//     Enc/Inputs/In/nState2 @bit 5 <-> ENC Status compact Channel 1/Status/Sync error
//     Enc/Inputs/In/nState2 @bit 5 <-> ENC Status compact Channel 2/Status/Sync error
//     Enc/Inputs/In/nState2 @bit 7 <-> ENC Status compact Channel 1/Status/TxPDO Toggle
//     Enc/Inputs/In/nState2 @bit 7 <-> ENC Status compact Channel 2/Status/TxPDO Toggle
//     Enc/Inputs/In/nState4 @bit 1 <-> WcState/InputToggle
//     Enc/Inputs/In/nState4 <-> WcState/WcState
//     Enc/Outputs/Out/nCtrl1 @bit 3 <-> ENC Control compact Channel 1/Control/Enable latch extern on negative edge
//     Enc/Outputs/Out/nCtrl1 @bit 3 <-> ENC Control compact Channel 2/Control/Enable latch extern on negative edge
//     Enc/Outputs/Out/nCtrl1 @bit 1 <-> ENC Control compact Channel 1/Control/Enable latch extern on positive edge
//     Enc/Outputs/Out/nCtrl1 @bit 1 <-> ENC Control compact Channel 2/Control/Enable latch extern on positive edge
//     Enc/Outputs/Out/nCtrl1 @bit 2 <-> ENC Control compact Channel 1/Control/Set counter
//     Enc/Outputs/Out/nCtrl1 @bit 2 <-> ENC Control compact Channel 2/Control/Set counter
//     Enc/Outputs/Out/nDataOut1[0] <-> ENC Control compact Channel 1/Set counter value
//     Enc/Outputs/Out/nDataOut1[0] <-> ENC Control compact Channel 2/Set counter value
//   NC-Task 1 SAF/Axes/Axis 1 <-> Long-CarryDrop (EtherCAT)/Long-Straight 1 (EP7342-0002)
//     Drive/Inputs/In/nState1 @bit 3 <-> DCM Status Channel 1/Status/Error
//     Drive/Inputs/In/nState1 @bit 5 <-> DCM Status Channel 1/Status/Moving negative
//     Drive/Inputs/In/nState1 @bit 4 <-> DCM Status Channel 1/Status/Moving positive
//     Drive/Inputs/In/nState1 @bit 1 <-> DCM Status Channel 1/Status/Ready
//     Drive/Inputs/In/nState1 <-> DCM Status Channel 1/Status/Ready to enable
//     Drive/Inputs/In/nState1 @bit 6 <-> DCM Status Channel 1/Status/Torque reduced
//     Drive/Inputs/In/nState1 @bit 2 <-> DCM Status Channel 1/Status/Warning
//     Drive/Inputs/In/nState2 @bit 3 <-> DCM Status Channel 1/Status/Digital input 1
//     Drive/Inputs/In/nState2 @bit 4 <-> DCM Status Channel 1/Status/Digital input 2
//     Drive/Inputs/In/nState2 @bit 5 <-> DCM Status Channel 1/Status/Sync error
//     Drive/Inputs/In/nState2 @bit 7 <-> DCM Status Channel 1/Status/TxPDO Toggle
//     Drive/Inputs/In/nState4 @bit 1 <-> WcState/InputToggle
//     Drive/Inputs/In/nState4 <-> WcState/WcState
//     Drive/Outputs/Out/nCtrl1 <-> DCM Control Channel 1/Control/Enable
//     Drive/Outputs/Out/nCtrl1 @bit 2 <-> DCM Control Channel 1/Control/Reduce torque
//     Drive/Outputs/Out/nCtrl1 @bit 1 <-> DCM Control Channel 1/Control/Reset
//     Drive/Outputs/Out/nDataOut2[0] <-> DCM Velocity Channel 1/Velocity
//     Enc/Inputs/In/nDataIn1[0] <-> ENC Status compact Channel 1/Counter value
//     Enc/Inputs/In/nDataIn2[0] <-> ENC Status compact Channel 1/Latch value
//     Enc/Inputs/In/nState1 @bit 4 <-> ENC Status compact Channel 1/Status/Counter overflow
//     Enc/Inputs/In/nState1 @bit 3 <-> ENC Status compact Channel 1/Status/Counter underflow
//     Enc/Inputs/In/nState1 @bit 7 <-> ENC Status compact Channel 1/Status/Extrapolation stall
//     Enc/Inputs/In/nState1 @bit 1 <-> ENC Status compact Channel 1/Status/Latch extern valid
//     Enc/Inputs/In/nState1 @bit 2 <-> ENC Status compact Channel 1/Status/Set counter done
//     Enc/Inputs/In/nState2 @bit 4 <-> ENC Status compact Channel 1/Status/Status of extern latch
//     Enc/Inputs/In/nState2 <-> ENC Status compact Channel 1/Status/Status of input A
//     Enc/Inputs/In/nState2 @bit 1 <-> ENC Status compact Channel 1/Status/Status of input B
//     Enc/Inputs/In/nState2 @bit 5 <-> ENC Status compact Channel 1/Status/Sync error
//     Enc/Inputs/In/nState2 @bit 7 <-> ENC Status compact Channel 1/Status/TxPDO Toggle
//     Enc/Inputs/In/nState4 @bit 1 <-> WcState/InputToggle
//     Enc/Inputs/In/nState4 <-> WcState/WcState
//     Enc/Outputs/Out/nCtrl1 @bit 3 <-> ENC Control compact Channel 1/Control/Enable latch extern on negative edge
//     Enc/Outputs/Out/nCtrl1 @bit 1 <-> ENC Control compact Channel 1/Control/Enable latch extern on positive edge
//     Enc/Outputs/Out/nCtrl1 @bit 2 <-> ENC Control compact Channel 1/Control/Set counter
//     Enc/Outputs/Out/nDataOut1[0] <-> ENC Control compact Channel 1/Set counter value
//   NC-Task 1 SAF/Axes/Axis 1 <-> Untitled1/Untitled1 Instance
//     Inputs/FromPlc <-> PlcTask Outputs/MAIN.stAxis1.PlcToNc
//     Outputs/ToPlc <-> PlcTask Inputs/MAIN.stAxis1.NcToPlc
//   NC-Task 1 SAF/Axes/Axis 2 <-> Long-CarryDrop (EtherCAT)/Long-Straight 1 (EP7342-0002)
//     Drive/Inputs/In/nState1 @bit 3 <-> DCM Status Channel 2/Status/Error
//     Drive/Inputs/In/nState1 @bit 5 <-> DCM Status Channel 2/Status/Moving negative
//     Drive/Inputs/In/nState1 @bit 4 <-> DCM Status Channel 2/Status/Moving positive
//     Drive/Inputs/In/nState1 @bit 1 <-> DCM Status Channel 2/Status/Ready
//     Drive/Inputs/In/nState1 <-> DCM Status Channel 2/Status/Ready to enable
//     Drive/Inputs/In/nState1 @bit 6 <-> DCM Status Channel 2/Status/Torque reduced
//     Drive/Inputs/In/nState1 @bit 2 <-> DCM Status Channel 2/Status/Warning
//     Drive/Inputs/In/nState2 @bit 3 <-> DCM Status Channel 2/Status/Digital input 1
//     Drive/Inputs/In/nState2 @bit 4 <-> DCM Status Channel 2/Status/Digital input 2
//     Drive/Inputs/In/nState2 @bit 5 <-> DCM Status Channel 2/Status/Sync error
//     Drive/Inputs/In/nState2 @bit 7 <-> DCM Status Channel 2/Status/TxPDO Toggle
//     Drive/Inputs/In/nState4 @bit 1 <-> WcState/InputToggle
//     Drive/Inputs/In/nState4 <-> WcState/WcState
//     Drive/Outputs/Out/nCtrl1 <-> DCM Control Channel 2/Control/Enable
//     Drive/Outputs/Out/nCtrl1 @bit 2 <-> DCM Control Channel 2/Control/Reduce torque
//     Drive/Outputs/Out/nCtrl1 @bit 1 <-> DCM Control Channel 2/Control/Reset
//     Drive/Outputs/Out/nDataOut2[0] <-> DCM Velocity Channel 2/Velocity
//     Enc/Inputs/In/nDataIn1[0] <-> ENC Status compact Channel 2/Counter value
//     Enc/Inputs/In/nDataIn2[0] <-> ENC Status compact Channel 2/Latch value
//     Enc/Inputs/In/nState1 @bit 4 <-> ENC Status compact Channel 2/Status/Counter overflow
//     Enc/Inputs/In/nState1 @bit 3 <-> ENC Status compact Channel 2/Status/Counter underflow
//     Enc/Inputs/In/nState1 @bit 7 <-> ENC Status compact Channel 2/Status/Extrapolation stall
//     Enc/Inputs/In/nState1 @bit 1 <-> ENC Status compact Channel 2/Status/Latch extern valid
//     Enc/Inputs/In/nState1 @bit 2 <-> ENC Status compact Channel 2/Status/Set counter done
//     Enc/Inputs/In/nState2 @bit 4 <-> ENC Status compact Channel 2/Status/Status of extern latch
//     Enc/Inputs/In/nState2 <-> ENC Status compact Channel 2/Status/Status of input A
//     Enc/Inputs/In/nState2 @bit 1 <-> ENC Status compact Channel 2/Status/Status of input B
//     Enc/Inputs/In/nState2 @bit 5 <-> ENC Status compact Channel 2/Status/Sync error
//     Enc/Inputs/In/nState2 @bit 7 <-> ENC Status compact Channel 2/Status/TxPDO Toggle
//     Enc/Inputs/In/nState4 @bit 1 <-> WcState/InputToggle
//     Enc/Inputs/In/nState4 <-> WcState/WcState
//     Enc/Outputs/Out/nCtrl1 @bit 3 <-> ENC Control compact Channel 2/Control/Enable latch extern on negative edge
//     Enc/Outputs/Out/nCtrl1 @bit 1 <-> ENC Control compact Channel 2/Control/Enable latch extern on positive edge
//     Enc/Outputs/Out/nCtrl1 @bit 2 <-> ENC Control compact Channel 2/Control/Set counter
//     Enc/Outputs/Out/nDataOut1[0] <-> ENC Control compact Channel 2/Set counter value
//   NC-Task 1 SAF/Axes/Axis 2 <-> Untitled1/Untitled1 Instance
//     Inputs/FromPlc <-> PlcTask Outputs/MAIN.stAxis2.PlcToNc
//     Outputs/ToPlc <-> PlcTask Inputs/MAIN.stAxis2.NcToPlc
//   NC-Task 1 SAF/Axes/Axis 3 <-> Long-CarryDrop (EtherCAT)/Long-Straight 2 (EP7342-0002)
//     Drive/Inputs/In/nState1 @bit 3 <-> DCM Status Channel 1/Status/Error
//     Drive/Inputs/In/nState1 @bit 5 <-> DCM Status Channel 1/Status/Moving negative
//     Drive/Inputs/In/nState1 @bit 4 <-> DCM Status Channel 1/Status/Moving positive
//     Drive/Inputs/In/nState1 @bit 1 <-> DCM Status Channel 1/Status/Ready
//     Drive/Inputs/In/nState1 <-> DCM Status Channel 1/Status/Ready to enable
//     Drive/Inputs/In/nState1 @bit 6 <-> DCM Status Channel 1/Status/Torque reduced
//     Drive/Inputs/In/nState1 @bit 2 <-> DCM Status Channel 1/Status/Warning
//     Drive/Inputs/In/nState2 @bit 3 <-> DCM Status Channel 1/Status/Digital input 1
//     Drive/Inputs/In/nState2 @bit 4 <-> DCM Status Channel 1/Status/Digital input 2
//     Drive/Inputs/In/nState2 @bit 5 <-> DCM Status Channel 1/Status/Sync error
//     Drive/Inputs/In/nState2 @bit 7 <-> DCM Status Channel 1/Status/TxPDO Toggle
//     Drive/Inputs/In/nState4 @bit 1 <-> WcState/InputToggle
//     Drive/Inputs/In/nState4 <-> WcState/WcState
//     Drive/Outputs/Out/nCtrl1 <-> DCM Control Channel 1/Control/Enable
//     Drive/Outputs/Out/nCtrl1 @bit 2 <-> DCM Control Channel 1/Control/Reduce torque
//     Drive/Outputs/Out/nCtrl1 @bit 1 <-> DCM Control Channel 1/Control/Reset
//     Drive/Outputs/Out/nDataOut2[0] <-> DCM Velocity Channel 1/Velocity
//     Enc/Inputs/In/nDataIn1[0] <-> ENC Status compact Channel 1/Counter value
//     Enc/Inputs/In/nDataIn2[0] <-> ENC Status compact Channel 1/Latch value
//     Enc/Inputs/In/nState1 @bit 4 <-> ENC Status compact Channel 1/Status/Counter overflow
//     Enc/Inputs/In/nState1 @bit 3 <-> ENC Status compact Channel 1/Status/Counter underflow
//     Enc/Inputs/In/nState1 @bit 7 <-> ENC Status compact Channel 1/Status/Extrapolation stall
//     Enc/Inputs/In/nState1 @bit 1 <-> ENC Status compact Channel 1/Status/Latch extern valid
//     Enc/Inputs/In/nState1 @bit 2 <-> ENC Status compact Channel 1/Status/Set counter done
//     Enc/Inputs/In/nState2 @bit 4 <-> ENC Status compact Channel 1/Status/Status of extern latch
//     Enc/Inputs/In/nState2 <-> ENC Status compact Channel 1/Status/Status of input A
//     Enc/Inputs/In/nState2 @bit 1 <-> ENC Status compact Channel 1/Status/Status of input B
//     Enc/Inputs/In/nState2 @bit 5 <-> ENC Status compact Channel 1/Status/Sync error
//     Enc/Inputs/In/nState2 @bit 7 <-> ENC Status compact Channel 1/Status/TxPDO Toggle
//     Enc/Inputs/In/nState4 @bit 1 <-> WcState/InputToggle
//     Enc/Inputs/In/nState4 <-> WcState/WcState
//     Enc/Outputs/Out/nCtrl1 @bit 3 <-> ENC Control compact Channel 1/Control/Enable latch extern on negative edge
//     Enc/Outputs/Out/nCtrl1 @bit 1 <-> ENC Control compact Channel 1/Control/Enable latch extern on positive edge
//     Enc/Outputs/Out/nCtrl1 @bit 2 <-> ENC Control compact Channel 1/Control/Set counter
//     Enc/Outputs/Out/nDataOut1[0] <-> ENC Control compact Channel 1/Set counter value
//   NC-Task 1 SAF/Axes/Axis 3 <-> Untitled1/Untitled1 Instance
//     Inputs/FromPlc <-> PlcTask Outputs/MAIN.stAxis3.PlcToNc
//     Outputs/ToPlc <-> PlcTask Inputs/MAIN.stAxis3.NcToPlc
//   NC-Task 1 SAF/Axes/Axis 4 <-> Long-CarryDrop (EtherCAT)/Long-Straight 2 (EP7342-0002)
//     Drive/Inputs/In/nState1 @bit 3 <-> DCM Status Channel 2/Status/Error
//     Drive/Inputs/In/nState1 @bit 5 <-> DCM Status Channel 2/Status/Moving negative
//     Drive/Inputs/In/nState1 @bit 4 <-> DCM Status Channel 2/Status/Moving positive
//     Drive/Inputs/In/nState1 @bit 1 <-> DCM Status Channel 2/Status/Ready
//     Drive/Inputs/In/nState1 <-> DCM Status Channel 2/Status/Ready to enable
//     Drive/Inputs/In/nState1 @bit 6 <-> DCM Status Channel 2/Status/Torque reduced
//     Drive/Inputs/In/nState1 @bit 2 <-> DCM Status Channel 2/Status/Warning
//     Drive/Inputs/In/nState2 @bit 3 <-> DCM Status Channel 2/Status/Digital input 1
//     Drive/Inputs/In/nState2 @bit 4 <-> DCM Status Channel 2/Status/Digital input 2
//     Drive/Inputs/In/nState2 @bit 5 <-> DCM Status Channel 2/Status/Sync error
//     Drive/Inputs/In/nState2 @bit 7 <-> DCM Status Channel 2/Status/TxPDO Toggle
//     Drive/Inputs/In/nState4 @bit 1 <-> WcState/InputToggle
//     Drive/Inputs/In/nState4 <-> WcState/WcState
//     Drive/Outputs/Out/nCtrl1 <-> DCM Control Channel 2/Control/Enable
//     Drive/Outputs/Out/nCtrl1 @bit 2 <-> DCM Control Channel 2/Control/Reduce torque
//     Drive/Outputs/Out/nCtrl1 @bit 1 <-> DCM Control Channel 2/Control/Reset
//     Drive/Outputs/Out/nDataOut2[0] <-> DCM Velocity Channel 2/Velocity
//     Enc/Inputs/In/nDataIn1[0] <-> ENC Status compact Channel 2/Counter value
//     Enc/Inputs/In/nDataIn2[0] <-> ENC Status compact Channel 2/Latch value
//     Enc/Inputs/In/nState1 @bit 4 <-> ENC Status compact Channel 2/Status/Counter overflow
//     Enc/Inputs/In/nState1 @bit 3 <-> ENC Status compact Channel 2/Status/Counter underflow
//     Enc/Inputs/In/nState1 @bit 7 <-> ENC Status compact Channel 2/Status/Extrapolation stall
//     Enc/Inputs/In/nState1 @bit 1 <-> ENC Status compact Channel 2/Status/Latch extern valid
//     Enc/Inputs/In/nState1 @bit 2 <-> ENC Status compact Channel 2/Status/Set counter done
//     Enc/Inputs/In/nState2 @bit 4 <-> ENC Status compact Channel 2/Status/Status of extern latch
//     Enc/Inputs/In/nState2 <-> ENC Status compact Channel 2/Status/Status of input A
//     Enc/Inputs/In/nState2 @bit 1 <-> ENC Status compact Channel 2/Status/Status of input B
//     Enc/Inputs/In/nState2 @bit 5 <-> ENC Status compact Channel 2/Status/Sync error
//     Enc/Inputs/In/nState2 @bit 7 <-> ENC Status compact Channel 2/Status/TxPDO Toggle
//     Enc/Inputs/In/nState4 @bit 1 <-> WcState/InputToggle
//     Enc/Inputs/In/nState4 <-> WcState/WcState
//     Enc/Outputs/Out/nCtrl1 @bit 3 <-> ENC Control compact Channel 2/Control/Enable latch extern on negative edge
//     Enc/Outputs/Out/nCtrl1 @bit 1 <-> ENC Control compact Channel 2/Control/Enable latch extern on positive edge
//     Enc/Outputs/Out/nCtrl1 @bit 2 <-> ENC Control compact Channel 2/Control/Set counter
//     Enc/Outputs/Out/nDataOut1[0] <-> ENC Control compact Channel 2/Set counter value
//   NC-Task 1 SAF/Axes/Axis 4 <-> Untitled1/Untitled1 Instance
//     Inputs/FromPlc <-> PlcTask Outputs/MAIN.stAxis4.PlcToNc
//     Outputs/ToPlc <-> PlcTask Inputs/MAIN.stAxis4.NcToPlc
//   NC-Task 1 SAF/Axes/Axis 5 <-> Long-CarryDrop (EtherCAT)/Short-Straight 1 (EP7342-0002)
//     Drive/Inputs/In/nState1 @bit 3 <-> DCM Status Channel 1/Status/Error
//     Drive/Inputs/In/nState1 @bit 5 <-> DCM Status Channel 1/Status/Moving negative
//     Drive/Inputs/In/nState1 @bit 4 <-> DCM Status Channel 1/Status/Moving positive
//     Drive/Inputs/In/nState1 @bit 1 <-> DCM Status Channel 1/Status/Ready
//     Drive/Inputs/In/nState1 <-> DCM Status Channel 1/Status/Ready to enable
//     Drive/Inputs/In/nState1 @bit 6 <-> DCM Status Channel 1/Status/Torque reduced
//     Drive/Inputs/In/nState1 @bit 2 <-> DCM Status Channel 1/Status/Warning
//     Drive/Inputs/In/nState2 @bit 3 <-> DCM Status Channel 1/Status/Digital input 1
//     Drive/Inputs/In/nState2 @bit 4 <-> DCM Status Channel 1/Status/Digital input 2
//     Drive/Inputs/In/nState2 @bit 5 <-> DCM Status Channel 1/Status/Sync error
//     Drive/Inputs/In/nState2 @bit 7 <-> DCM Status Channel 1/Status/TxPDO Toggle
//     Drive/Inputs/In/nState4 @bit 1 <-> WcState/InputToggle
//     Drive/Inputs/In/nState4 <-> WcState/WcState
//     Drive/Outputs/Out/nCtrl1 <-> DCM Control Channel 1/Control/Enable
//     Drive/Outputs/Out/nCtrl1 @bit 2 <-> DCM Control Channel 1/Control/Reduce torque
//     Drive/Outputs/Out/nCtrl1 @bit 1 <-> DCM Control Channel 1/Control/Reset
//     Drive/Outputs/Out/nDataOut2[0] <-> DCM Velocity Channel 1/Velocity
//     Enc/Inputs/In/nDataIn1[0] <-> ENC Status compact Channel 1/Counter value
//     Enc/Inputs/In/nDataIn2[0] <-> ENC Status compact Channel 1/Latch value
//     Enc/Inputs/In/nState1 @bit 4 <-> ENC Status compact Channel 1/Status/Counter overflow
//     Enc/Inputs/In/nState1 @bit 3 <-> ENC Status compact Channel 1/Status/Counter underflow
//     Enc/Inputs/In/nState1 @bit 7 <-> ENC Status compact Channel 1/Status/Extrapolation stall
//     Enc/Inputs/In/nState1 @bit 1 <-> ENC Status compact Channel 1/Status/Latch extern valid
//     Enc/Inputs/In/nState1 @bit 2 <-> ENC Status compact Channel 1/Status/Set counter done
//     Enc/Inputs/In/nState2 @bit 4 <-> ENC Status compact Channel 1/Status/Status of extern latch
//     Enc/Inputs/In/nState2 <-> ENC Status compact Channel 1/Status/Status of input A
//     Enc/Inputs/In/nState2 @bit 1 <-> ENC Status compact Channel 1/Status/Status of input B
//     Enc/Inputs/In/nState2 @bit 5 <-> ENC Status compact Channel 1/Status/Sync error
//     Enc/Inputs/In/nState2 @bit 7 <-> ENC Status compact Channel 1/Status/TxPDO Toggle
//     Enc/Inputs/In/nState4 @bit 1 <-> WcState/InputToggle
//     Enc/Inputs/In/nState4 <-> WcState/WcState
//     Enc/Outputs/Out/nCtrl1 @bit 3 <-> ENC Control compact Channel 1/Control/Enable latch extern on negative edge
//     Enc/Outputs/Out/nCtrl1 @bit 1 <-> ENC Control compact Channel 1/Control/Enable latch extern on positive edge
//     Enc/Outputs/Out/nCtrl1 @bit 2 <-> ENC Control compact Channel 1/Control/Set counter
//     Enc/Outputs/Out/nDataOut1[0] <-> ENC Control compact Channel 1/Set counter value
//   NC-Task 1 SAF/Axes/Axis 5 <-> Untitled1/Untitled1 Instance
//     Inputs/FromPlc <-> PlcTask Outputs/MAIN.stAxis5.PlcToNc
//     Outputs/ToPlc <-> PlcTask Inputs/MAIN.stAxis5.NcToPlc
//   NC-Task 1 SAF/Axes/Axis 6 <-> Long-CarryDrop (EtherCAT)/Short-Straight 1 (EP7342-0002)
//     Drive/Inputs/In/nState1 @bit 3 <-> DCM Status Channel 2/Status/Error
//     Drive/Inputs/In/nState1 @bit 5 <-> DCM Status Channel 2/Status/Moving negative
//     Drive/Inputs/In/nState1 @bit 4 <-> DCM Status Channel 2/Status/Moving positive
//     Drive/Inputs/In/nState1 @bit 1 <-> DCM Status Channel 2/Status/Ready
//     Drive/Inputs/In/nState1 <-> DCM Status Channel 2/Status/Ready to enable
//     Drive/Inputs/In/nState1 @bit 6 <-> DCM Status Channel 2/Status/Torque reduced
//     Drive/Inputs/In/nState1 @bit 2 <-> DCM Status Channel 2/Status/Warning
//     Drive/Inputs/In/nState2 @bit 3 <-> DCM Status Channel 2/Status/Digital input 1
//     Drive/Inputs/In/nState2 @bit 4 <-> DCM Status Channel 2/Status/Digital input 2
//     Drive/Inputs/In/nState2 @bit 5 <-> DCM Status Channel 2/Status/Sync error
//     Drive/Inputs/In/nState2 @bit 7 <-> DCM Status Channel 2/Status/TxPDO Toggle
//     Drive/Inputs/In/nState4 @bit 1 <-> WcState/InputToggle
//     Drive/Inputs/In/nState4 <-> WcState/WcState
//     Drive/Outputs/Out/nCtrl1 <-> DCM Control Channel 2/Control/Enable
//     Drive/Outputs/Out/nCtrl1 @bit 2 <-> DCM Control Channel 2/Control/Reduce torque
//     Drive/Outputs/Out/nCtrl1 @bit 1 <-> DCM Control Channel 2/Control/Reset
//     Drive/Outputs/Out/nDataOut2[0] <-> DCM Velocity Channel 2/Velocity
//     Enc/Inputs/In/nDataIn1[0] <-> ENC Status compact Channel 2/Counter value
//     Enc/Inputs/In/nDataIn2[0] <-> ENC Status compact Channel 2/Latch value
//     Enc/Inputs/In/nState1 @bit 4 <-> ENC Status compact Channel 2/Status/Counter overflow
//     Enc/Inputs/In/nState1 @bit 3 <-> ENC Status compact Channel 2/Status/Counter underflow
//     Enc/Inputs/In/nState1 @bit 7 <-> ENC Status compact Channel 2/Status/Extrapolation stall
//     Enc/Inputs/In/nState1 @bit 1 <-> ENC Status compact Channel 2/Status/Latch extern valid
//     Enc/Inputs/In/nState1 @bit 2 <-> ENC Status compact Channel 2/Status/Set counter done
//     Enc/Inputs/In/nState2 @bit 4 <-> ENC Status compact Channel 2/Status/Status of extern latch
//     Enc/Inputs/In/nState2 <-> ENC Status compact Channel 2/Status/Status of input A
//     Enc/Inputs/In/nState2 @bit 1 <-> ENC Status compact Channel 2/Status/Status of input B
//     Enc/Inputs/In/nState2 @bit 5 <-> ENC Status compact Channel 2/Status/Sync error
//     Enc/Inputs/In/nState2 @bit 7 <-> ENC Status compact Channel 2/Status/TxPDO Toggle
//     Enc/Inputs/In/nState4 @bit 1 <-> WcState/InputToggle
//     Enc/Inputs/In/nState4 <-> WcState/WcState
//     Enc/Outputs/Out/nCtrl1 @bit 3 <-> ENC Control compact Channel 2/Control/Enable latch extern on negative edge
//     Enc/Outputs/Out/nCtrl1 @bit 1 <-> ENC Control compact Channel 2/Control/Enable latch extern on positive edge
//     Enc/Outputs/Out/nCtrl1 @bit 2 <-> ENC Control compact Channel 2/Control/Set counter
//     Enc/Outputs/Out/nDataOut1[0] <-> ENC Control compact Channel 2/Set counter value
//   NC-Task 1 SAF/Axes/Axis 6 <-> Untitled1/Untitled1 Instance
//     Inputs/FromPlc <-> PlcTask Outputs/MAIN.stAxis6.PlcToNc
//     Outputs/ToPlc <-> PlcTask Inputs/MAIN.stAxis6.NcToPlc
//   NC-Task 1 SAF/Axes/Axis 7 <-> Long-CarryDrop (EtherCAT)/Incline-Belt 1 (EP7041-0002)
//     Drive/Inputs/In/nState1 @bit 3 <-> STM Status/Status/Error
//     Drive/Inputs/In/nState1 @bit 5 <-> STM Status/Status/Moving negative
//     Drive/Inputs/In/nState1 @bit 4 <-> STM Status/Status/Moving positive
//     Drive/Inputs/In/nState1 @bit 1 <-> STM Status/Status/Ready
//     Drive/Inputs/In/nState1 <-> STM Status/Status/Ready to enable
//     Drive/Inputs/In/nState1 @bit 6 <-> STM Status/Status/Torque reduced
//     Drive/Inputs/In/nState1 @bit 2 <-> STM Status/Status/Warning
//     Drive/Inputs/In/nState2 @bit 3 <-> STM Status/Status/Digital input 1
//     Drive/Inputs/In/nState2 @bit 4 <-> STM Status/Status/Digital input 2
//     Drive/Inputs/In/nState2 @bit 5 <-> STM Status/Status/Sync error
//     Drive/Inputs/In/nState2 @bit 7 <-> STM Status/Status/TxPDO Toggle
//     Drive/Inputs/In/nState4 @bit 1 <-> WcState/InputToggle
//     Drive/Inputs/In/nState4 <-> WcState/WcState
//     Drive/Outputs/Out/nCtrl1 <-> STM Control/Control/Enable
//     Drive/Outputs/Out/nCtrl1 @bit 2 <-> STM Control/Control/Reduce torque
//     Drive/Outputs/Out/nCtrl1 @bit 1 <-> STM Control/Control/Reset
//     Drive/Outputs/Out/nCtrl2 @bit 3 <-> STM Control/Control/Digital output 1
//     Drive/Outputs/Out/nDataOut2[0] <-> STM Velocity/Velocity
//     Enc/Inputs/In/nDataIn1[0] <-> ENC Status compact/Counter value
//     Enc/Inputs/In/nDataIn2[0] <-> ENC Status compact/Latch value
//     Enc/Inputs/In/nState1 @bit 4 <-> ENC Status compact/Status/Counter overflow
//     Enc/Inputs/In/nState1 @bit 3 <-> ENC Status compact/Status/Counter underflow
//     Enc/Inputs/In/nState1 @bit 7 <-> ENC Status compact/Status/Extrapolation stall
//     Enc/Inputs/In/nState1 <-> ENC Status compact/Status/Latch C valid
//     Enc/Inputs/In/nState1 @bit 1 <-> ENC Status compact/Status/Latch extern valid
//     Enc/Inputs/In/nState1 @bit 2 <-> ENC Status compact/Status/Set counter done
//     Enc/Inputs/In/nState2 @bit 4 <-> ENC Status compact/Status/Status of extern latch
//     Enc/Inputs/In/nState2 <-> ENC Status compact/Status/Status of input A
//     Enc/Inputs/In/nState2 @bit 1 <-> ENC Status compact/Status/Status of input B
//     Enc/Inputs/In/nState2 @bit 2 <-> ENC Status compact/Status/Status of input C
//     Enc/Inputs/In/nState2 @bit 5 <-> ENC Status compact/Status/Sync error
//     Enc/Inputs/In/nState2 @bit 7 <-> ENC Status compact/Status/TxPDO Toggle
//     Enc/Inputs/In/nState4 @bit 1 <-> WcState/InputToggle
//     Enc/Inputs/In/nState4 <-> WcState/WcState
//     Enc/Outputs/Out/nCtrl1 <-> ENC Control compact/Control/Enable latch C
//     Enc/Outputs/Out/nCtrl1 @bit 3 <-> ENC Control compact/Control/Enable latch extern on negative edge
//     Enc/Outputs/Out/nCtrl1 @bit 1 <-> ENC Control compact/Control/Enable latch extern on positive edge
//     Enc/Outputs/Out/nCtrl1 @bit 2 <-> ENC Control compact/Control/Set counter
//     Enc/Outputs/Out/nDataOut1[0] <-> ENC Control compact/Set counter value
//   NC-Task 1 SAF/Axes/Axis 7 <-> Untitled1/Untitled1 Instance
//     Inputs/FromPlc <-> PlcTask Outputs/MAIN.stAxis7.PlcToNc
//     Outputs/ToPlc <-> PlcTask Inputs/MAIN.stAxis7.NcToPlc

CONFIGURATION Untitled1
    RESOURCE PLC ON TwinCAT3
        TASK PlcTask(INTERVAL := T#10ms, PRIORITY := 20);
        PROGRAM MAIN WITH PlcTask : MAIN;
    END_RESOURCE
END_CONFIGURATION

// ---- DUTs/EP7402_REF.TcDUT

TYPE EP7402_REF :
STRUCT
	stInputs	AT %I* : ARRAY[0..7] OF BYTE;//MDR_CONTROL.EP7402_Inputs;
	stOutputs	AT %Q* : ARRAY[0..7] OF BYTE;//MDR_Control.EP7402_Outputs;
END_STRUCT
END_TYPE

// ---- GVLs/Global_Constants.TcGVL
{attribute 'qualified_only'}
VAR_GLOBAL CONSTANT
	nMAXGroups	: UINT := 2;
END_VAR

// ---- GVLs/GVL_IO.TcGVL
{attribute 'qualified_only'}
VAR_GLOBAL
	arrId	AT %I*:	ARRAY[0..255] OF UINT;
END_VAR

// ---- POUs/Interfaces/I_ControlScheme.TcIO
INTERFACE I_ControlScheme

END_INTERFACE

// ---- POUs/Interfaces/I_Conveyer.TcIO
INTERFACE I_Conveyer

METHOD Execute : BOOL
VAR_INPUT
END_VAR
END_METHOD

METHOD Reset : BOOL
VAR_INPUT
END_VAR
END_METHOD

METHOD Start : BOOL
VAR_INPUT
END_VAR
END_METHOD

METHOD Stop : BOOL
VAR_INPUT
END_VAR
END_METHOD

END_INTERFACE

// ---- POUs/Interfaces/I_MDRConveyer.TcIO
INTERFACE I_MDRConveyer EXTENDS I_Conveyer

PROPERTY MDRController : EP7402_REF
GET
END_GET
SET
END_SET
END_PROPERTY

END_INTERFACE

// ---- POUs/Interfaces/I_NcConveyer.TcIO
INTERFACE I_NcConveyer EXTENDS I_Conveyer

PROPERTY Axis1 : AXIS_REF
GET
END_GET
SET
END_SET
END_PROPERTY

PROPERTY Axis2 : AXIS_REF
GET
END_GET
SET
END_SET
END_PROPERTY

END_INTERFACE

// ---- POUs/MAIN.TcPOU
PROGRAM MAIN
VAR
	{IF defined (Variant3)}
	stAxis1	: EP7402_REF;
	stAxis2	: EP7402_REF;
	stAxis3	: EP7402_REF;
	
	{ELSE}
	stAxis1	: AXIS_REF;
	stAxis2	: AXIS_REF;
	stAxis3	: AXIS_REF;
	stAxis4	: AXIS_REF;
	{END_IF}
	{IF defined (Group1)}
	stAxis5	: AXIS_REF;
	stAxis6	: AXIS_REF;
	stAxis7	: AXIS_REF;
	stAxis8	: AXIS_REF;
	{END_IF}
	
	(*{IF defined (Variant1)}
	FB_ConveyerSequence	:	FB_LongCarryDrop;
	{ELSIF defined (Variant2)}
	FB_ConveyerSequence	:	FB_CarryDrop(Axis1 := stAxis1,Axis2 := stAxis2,Axis3 := stAxis3, Axis4 :=stAxis4);
	{ELSIF defined (Variant3)}
	FB_ConveyerSequence :	FB_LongTransfer(Axis1 := stAxis1,Axis2 := stAxis2,Axis3 := stAxis3);;
	{ELSE}
	FB_ConveyerSequence	:	FB_CarryDrop(Axis1 := stAxis1, Axis2 := stAxis2, Axis3 := stAxis3, Axis4 :=stAxis4, Axis5 := stAxis5, Axis6 := stAxis6, Axis7 := stAxis7, Axis8 := stAxis8);
	{END_IF}
*)
END_VAR

END_PROGRAM

// ---- POUs/Function Blocks/ControlSchemes/FB_LongCarryDrop.TcPOU
FUNCTION_BLOCK FB_LongCarryDrop IMPLEMENTS I_ControlScheme
VAR_INPUT
END_VAR
VAR_OUTPUT
END_VAR
VAR
	fbLongStraight1	: FB_LsNcConveyer;
	fbLongStraight2	: FB_LsNcConveyer;
	fbIncline		: FB_InclineNcConveyer;
	fbShortStraight	: FB_SsNcConveyer;
	nState 	: INT := 0;
END_VAR
VAR_IN_OUT
	Axis1	: AXIS_REF;
	Axis2	: AXIS_REF;
	Axis3	: AXIS_REF;
	Axis4	: AXIS_REF;
	Axis5	: AXIS_REF;
	Axis6	: AXIS_REF;
	Axis7	: AXIS_REF;
	Axis8	: AXIS_REF; 
END_VAR

CASE nState OF
0:
	//TODO:Assign Axes
	nState :=1;
1: 
	fbLongStraight1.Start();
	fbLongStraight2.Start();
	fbIncline.Start();
	fbShortStraight.Start();
	
	
2:
	fbLongStraight1.Execute();
	fbLongStraight2.Execute();
	fbIncline.Execute();
	fbShortStraight.Execute();

	nState := 3;
3:
	//TO-DO call Stop methods
	nState := 4;
4:
	//TODO: call Reset methods
END_CASE

END_FUNCTION_BLOCK

// ---- POUs/Function Blocks/NcConveyers/FB_LsNcConveyer.TcPOU
FUNCTION_BLOCK FB_LsNcConveyer IMPLEMENTS  I_NcConveyer
VAR_INPUT
END_VAR
VAR_OUTPUT
END_VAR
VAR
	_Axis1	: AXIS_REF;
	_Axis2	: AXIS_REF;
END_VAR

{warning 'add property implementation'}
PROPERTY Axis1 : Tc2_MC2.AXIS_REF
GET
Axis1 := _Axis1;
END_GET
SET
_Axis1 := Axis1;
END_SET
END_PROPERTY

{warning 'add property implementation'}
PROPERTY Axis2 : Tc2_MC2.AXIS_REF
GET
Axis2 := _Axis2;
END_GET
SET
_Axis2 := Axis2;
END_SET
END_PROPERTY

{warning 'add method implementation '}
METHOD Execute : BOOL
ADSLOGSTR(ADSLOG_MSGTYPE_LOG,'Moving Long-Straight','');
END_METHOD

{warning 'add method implementation '}
METHOD Reset : BOOL
ADSLOGSTR(ADSLOG_MSGTYPE_LOG,'Reseting Long-Straight','');
END_METHOD

{warning 'add method implementation '}
METHOD Start : BOOL
ADSLOGSTR(ADSLOG_MSGTYPE_LOG,'Powering on Long-Straight','');
END_METHOD

{warning 'add method implementation '}
METHOD Stop : BOOL
ADSLOGSTR(ADSLOG_MSGTYPE_LOG,'Stopping Long-Straight','');
END_METHOD

END_FUNCTION_BLOCK

// ---- POUs/Function Blocks/NcConveyers/FB_InclineNcConveyer.TcPOU
FUNCTION_BLOCK FB_InclineNcConveyer IMPLEMENTS  I_NcConveyer
VAR_INPUT
END_VAR
VAR_OUTPUT
END_VAR
VAR
	_Axis1	: AXIS_REF;
	_Axis2	: AXIS_REF;
	
END_VAR

{warning 'add property implementation'}
PROPERTY Axis1 : Tc2_MC2.AXIS_REF
GET
Axis1 := _Axis1;
END_GET
SET
_Axis1 := Axis1;
END_SET
END_PROPERTY

{warning 'add property implementation'}
PROPERTY Axis2 : Tc2_MC2.AXIS_REF
GET
Axis2 := _Axis2;
END_GET
SET
_Axis2 := Axis2;
END_SET
END_PROPERTY

{warning 'add method implementation '}
METHOD Execute : BOOL
ADSLOGSTR(ADSLOG_MSGTYPE_LOG,'Moving Incline-Belt','');
END_METHOD

{warning 'add method implementation '}
METHOD Reset : BOOL
ADSLOGSTR(ADSLOG_MSGTYPE_LOG,'Reseting Incline-Belt','');
END_METHOD

{warning 'add method implementation '}
METHOD Start : BOOL
ADSLOGSTR(ADSLOG_MSGTYPE_LOG,'Powering Incline-Belt on','');
END_METHOD

{warning 'add method implementation '}
METHOD Stop : BOOL
ADSLOGSTR(ADSLOG_MSGTYPE_LOG,'Stopping Incline-Belt','');
END_METHOD

END_FUNCTION_BLOCK

// ---- POUs/Function Blocks/NcConveyers/FB_SsNcConveyer.TcPOU
FUNCTION_BLOCK FB_SsNcConveyer IMPLEMENTS I_NcConveyer
VAR_INPUT
END_VAR
VAR_OUTPUT
END_VAR
VAR
	_Axis1	: AXIS_REF;
	_Axis2	: AXIS_REF;
	
END_VAR


PROPERTY Axis1 : Tc2_MC2.AXIS_REF
GET
Axis1 := _Axis1;
END_GET
SET
_Axis1 := Axis1;
END_SET
END_PROPERTY

PROPERTY Axis2 : Tc2_MC2.AXIS_REF
GET
Axis2 := _Axis2;
END_GET
SET
_Axis2 := Axis2;
END_SET
END_PROPERTY

METHOD Execute : BOOL
ADSLOGSTR(ADSLOG_MSGTYPE_LOG,'Moving short-straight','');
END_METHOD


METHOD Reset : BOOL
ADSLOGSTR(ADSLOG_MSGTYPE_LOG,'Reseting short-straight','');
END_METHOD

METHOD Start : BOOL
ADSLOGSTR(ADSLOG_MSGTYPE_LOG,'Powering Short-Straight on','');
END_METHOD

METHOD Stop : BOOL
ADSLOGSTR(ADSLOG_MSGTYPE_LOG,'Stopping short-straight','');
END_METHOD

END_FUNCTION_BLOCK

// ---- POUs/Function Blocks/ControlSchemes/FB_CarryDrop.TcPOU
FUNCTION_BLOCK FB_CarryDrop IMPLEMENTS I_ControlScheme
VAR_INPUT
END_VAR
VAR_OUTPUT
END_VAR
VAR
	fbIncline		: FB_InclineNcConveyer;
	fbShortStraight	: FB_SsNcConveyer;
	{IF defined (Group1)}
	fbShortStraight2	: FB_SsNcConveyer;
	fbDecline		: FB_DeclineNcConveyer;
	{END_IF}
	
	nState	: INT := 0;
END_VAR
VAR_IN_OUT
	Axis1	: AXIS_REF;
	Axis2	: AXIS_REF;
	Axis3	: AXIS_REF;
	Axis4	: AXIS_REF;
	{IF defined (group1)}
	Axis5	: AXIS_REF;
	Axis6	: AXIS_REF;
	Axis7	: AXIS_REF;
	Axis8	: AXIS_REF;
	{END_IF}
END_VAR

CASE nState OF
0:
	//TODO:Assign Axes
	nState :=1;
1: 
	fbIncline.Start();
	fbShortStraight.Start();
	{IF defined (Group1)}
	fbShortStraight2.Start();
	fbDecline.Start();
	{END_IF}
2:
	fbIncline.Execute();
	fbShortStraight.Execute();
	{IF defined (Group1)}
	fbShortStraight2.Execute();
	fbDecline.Execute();
	{END_IF}
	nState := 3;
3:
	//TO-DO call Stop methods
	nState := 4;
4:
	//TODO: call Reset methods
END_CASE

END_FUNCTION_BLOCK

// ---- POUs/Function Blocks/NcConveyers/FB_DeclineNcConveyer.TcPOU
FUNCTION_BLOCK FB_DeclineNcConveyer IMPLEMENTS  I_NcConveyer
VAR_INPUT
END_VAR
VAR_OUTPUT
END_VAR
VAR
	_Axis1	: AXIS_REF;
	_Axis2	: AXIS_REF;
	
END_VAR

{warning 'add property implementation'}
PROPERTY Axis1 : Tc2_MC2.AXIS_REF
GET
Axis1 := _Axis1;
END_GET
SET
_Axis1 := Axis1;
END_SET
END_PROPERTY

{warning 'add property implementation'}
PROPERTY Axis2 : Tc2_MC2.AXIS_REF
GET
Axis2 := _Axis2;
END_GET
SET
_Axis2 := Axis2;
END_SET
END_PROPERTY

{warning 'add method implementation '}
METHOD Execute : BOOL
ADSLOGSTR(ADSLOG_MSGTYPE_LOG,'Moving Decline-Belt','');
END_METHOD

{warning 'add method implementation '}
METHOD Reset : BOOL
ADSLOGSTR(ADSLOG_MSGTYPE_LOG,'Reseting Decline','');
END_METHOD

{warning 'add method implementation '}
METHOD Start : BOOL
ADSLOGSTR(ADSLOG_MSGTYPE_LOG,'Powering Decline-Belt On','');
END_METHOD

{warning 'add method implementation '}
METHOD Stop : BOOL
ADSLOGSTR(ADSLOG_MSGTYPE_LOG,'Stopping Decline-Belt','');
END_METHOD

END_FUNCTION_BLOCK

// ---- POUs/Function Blocks/ControlSchemes/FB_LongTransfer.TcPOU
FUNCTION_BLOCK FB_LongTransfer IMPLEMENTS I_ControlScheme
VAR_INPUT
END_VAR
VAR_OUTPUT
END_VAR
VAR
	fbDecline	: FB_DeclineMdrConveyer;
	fbLongStraight1		: FB_LsMdrConveyer;
	fbLongStraight2		: FB_LsMdrConveyer;
	nState: INT;
END_VAR
VAR_IN_OUT
	Axis1	:	EP7402_REF;
	Axis2	:	EP7402_REF;
	Axis3	:	EP7402_REF;
END_VAR

CASE nState OF
0:
	//TODO:Assign Axes
	nState :=1;
1: 
	fbLongStraight1.Start();
	fbLongStraight2.Start();
	fbDecline.Start();
	
	
	
2:
	fbLongStraight1.Execute();
	fbLongStraight2.Execute();
	fbDecline.Execute();
	

	nState := 3;
3:
	//TO-DO call Stop methods
	nState := 4;
4:
	//TODO: call Reset methods
END_CASE

END_FUNCTION_BLOCK

// ---- POUs/Function Blocks/MDRConveyers/FB_DeclineMdrConveyer.TcPOU
FUNCTION_BLOCK FB_DeclineMdrConveyer IMPLEMENTS  I_MDRConveyer
VAR_INPUT
END_VAR
VAR_OUTPUT
END_VAR
VAR
	_Controller	: EP7402_REF;

	
END_VAR

METHOD Execute : BOOL
ADSLOGSTR(ADSLOG_MSGTYPE_LOG,'Moving Long-Straight','');
END_METHOD


PROPERTY MDRController : EP7402_REF
GET
MDRController := _Controller;
END_GET
SET
_Controller := MDRController;
END_SET
END_PROPERTY


METHOD Reset : BOOL
ADSLOGSTR(ADSLOG_MSGTYPE_LOG,'Reseting Long-straight','');
END_METHOD


METHOD Start : BOOL
ADSLOGSTR(ADSLOG_MSGTYPE_LOG,'Powering on Long-straight','');
END_METHOD


METHOD Stop : BOOL
ADSLOGSTR(ADSLOG_MSGTYPE_LOG,'Stopping Long-straight','');
END_METHOD

END_FUNCTION_BLOCK

// ---- POUs/Function Blocks/MDRConveyers/FB_LsMdrConveyer.TcPOU
FUNCTION_BLOCK FB_LsMdrConveyer IMPLEMENTS  I_MDRConveyer
VAR_INPUT
END_VAR
VAR_OUTPUT
END_VAR
VAR
	_Controller	: EP7402_REF;

	
END_VAR


METHOD Execute : BOOL
ADSLOGSTR(ADSLOG_MSGTYPE_LOG,'Moving Long-Straight','');
END_METHOD

PROPERTY MDRController :EP7402_REF
GET
MDRController := _Controller;
END_GET
SET
_Controller := MDRController;
END_SET
END_PROPERTY


METHOD Reset : BOOL
ADSLOGSTR(ADSLOG_MSGTYPE_LOG,'Reseting Long-straight','');
END_METHOD


METHOD Start : BOOL
ADSLOGSTR(ADSLOG_MSGTYPE_LOG,'Powering on Long-straight','');
END_METHOD


METHOD Stop : BOOL
ADSLOGSTR(ADSLOG_MSGTYPE_LOG,'Stopping Long-straight','');
END_METHOD

END_FUNCTION_BLOCK

// ---- POUs/Function Blocks/HCGroupControl/FB_HotConnect1.TcPOU
FUNCTION_BLOCK FB_HotConnect1 IMPLEMENTS I_ControlScheme
VAR_INPUT
END_VAR
VAR_OUTPUT
END_VAR
VAR
	fbDecline1			: FB_DeclineNcConveyer;
	fbShortStraight1	: FB_SsNcConveyer;
	fbInline1			: FB_InclineNcConveyer;
END_VAR
VAR_IN_OUT
	Axis1	: AXIS_REF;
	Axis2	: AXIS_REF;
	Axis3	: AXIS_REF;
	Axis4	: AXIS_REF;
	Axis5	: AXIS_REF;
	Axis6	: AXIS_REF;
END_VAR

END_FUNCTION_BLOCK

// ---- POUs/Function Blocks/HCGroupControl/FB_HotConnect2.TcPOU
FUNCTION_BLOCK FB_HotConnect2
VAR_INPUT
END_VAR
VAR_OUTPUT
END_VAR
VAR
END_VAR

END_FUNCTION_BLOCK
